PROGRAM PULSE
VAR
	PULS1: TON;
	PULS2: TON;
	PULS3: TON;
	TP1: TP;
END_VAR

PULS1(IN:=TRUE,PT:=T#1MS);
SORTER_VAR.PULSE_OUT1 :=TP1.Q;
SORTER_VAR.PULSE_OUT2 :=TRUE;//NOT PULS1.Q;
TP1(IN:=PULS1.Q,PT:=T#1MS);
IF PULS1.Q THEN
	PULS2(IN:=TRUE,PT:=T#1MS);
END_IF
IF  PULS2.Q THEN
	PULS3(IN:=TRUE,PT:=T#1MS);
	PULS1(IN:=FALSE);
	PULS2(IN:=FALSE);
END_IF
(*
IF  PULS3.Q THEN
	PULS3(IN:=FALSE);
	PULS1(IN:=FALSE);
	PULS2(IN:=FALSE);
END_IF
*)

END_PROGRAM

(* stored: Version 1.1.0.1, ProductVersion 3.1.4020.12
   POU PULSE: Id {56e1537b-54bb-47b5-bc60-7fcbd60018d3}, SpecialFunc None *)
